INTERFACE I_Mc3AxisGear EXTENDS I_Base

METHOD GearIn
VAR_INPUT
END_VAR
END_METHOD

{attribute 'monitoring' := 'call'}
PROPERTY InGear : BOOL
GET
END_GET
END_PROPERTY

PROPERTY Master : I_Mc3Axis
SET
END_SET
END_PROPERTY

{attribute 'monitoring' := 'call'}
PROPERTY MasterHasError : BOOL
GET
END_GET
END_PROPERTY

{attribute 'monitoring' := 'call'}
PROPERTY RatioDenominator : LREAL
SET
END_SET
END_PROPERTY

{attribute 'monitoring' := 'call'}
PROPERTY RatioNumerator : LREAL
SET
END_SET
END_PROPERTY

PROPERTY ReactionToMasterError : EReactionToMasterError
SET
END_SET
END_PROPERTY

PROPERTY ReactionToSlaveError : EReactionToSlaveError
SET
END_SET
END_PROPERTY

END_INTERFACE

(* stored: Version 1.1.0.1, ProductVersion 3.1.4026.20
   Itf I_Mc3AxisGear: Id {d29e25bc-0997-4b31-a6fa-9701978da8b1}
   Method GearIn: Id {378a3fc8-f6d1-4f03-9d39-02b7fa888478}
   Property InGear: Id {477a68fb-b013-4f11-b369-e829532ccd42}
   Get Get: Id {0d83443b-d03c-49f4-af8f-d976f5920319}
   Property Master: Id {40f93b2a-edfa-450d-9f18-31964f978c98}
   Set Set: Id {8b8f6ac5-82f5-4ba2-85de-b9363b38e497}
   Property MasterHasError: Id {50a08d54-bdad-4d75-a2a1-99e068da0f00}
   Get Get: Id {a3ceb87e-40fa-49ae-802f-2ea6f87d2d36}
   Property RatioDenominator: Id {6c960b2d-55ca-4259-bab1-2bb43e8d3b26}
   Set Set: Id {f352ee05-edf1-46c9-9418-59d099d895a8}
   Property RatioNumerator: Id {40c83ab7-7a1a-46c5-b615-72864b70aaaf}
   Set Set: Id {b572cd86-f9d1-441a-8ae9-7582f49142d5}
   Property ReactionToMasterError: Id {d4d8710c-028b-4ec3-8577-b21f192ddb9d}
   Set Set: Id {080e3ee7-2f0a-4786-aebe-ee3a955ec697}
   Property ReactionToSlaveError: Id {8d086f56-f964-4b28-998e-30b6a17dc26c}
   Set Set: Id {bff48700-6202-4be6-8aeb-971b5950d703} *)
